INTERFACE I_MessageData

PROPERTY DirRoot : POINTER to string(255)
SET
END_SET
END_PROPERTY

PROPERTY ErrorIndex : reference to uint
SET
END_SET
END_PROPERTY

PROPERTY FileRoot : pointer to string(255)
SET
END_SET
END_PROPERTY

PROPERTY LocalTime : pointer to DT
SET
END_SET
END_PROPERTY

PROPERTY MessageIndex : reference to uint
SET
END_SET
END_PROPERTY

PROPERTY MsgList : pointer to ARRAY[1..GVL_MSG.MAX_MESSAGE] OF st_message
SET
END_SET
END_PROPERTY

END_INTERFACE

(* stored: Version 1.1.0.1
   Itf I_MessageData: Id {f6a96240-99ae-4618-b2ce-2104a304fee0}
   Property DirRoot: Id {caa07dbc-04ed-4392-a650-b335ab3d5005}
   Set Set: Id {fd0f934c-7d3d-4e0f-aecc-db828ecd61bd}
   Property ErrorIndex: Id {87d8f92c-f432-4c2d-b856-904c14d00dd3}
   Set Set: Id {18121a8a-40ab-41a6-b72d-61490f470a4a}
   Property FileRoot: Id {53c974bd-d010-4f69-a899-a1aaf707c45d}
   Set Set: Id {6ac54f9d-8006-4b91-9b1f-f40bcb34bbd2}
   Property LocalTime: Id {0ed9cddb-a9d3-4c4f-937d-34752c417a65}
   Set Set: Id {6a30d4b9-5ac5-49e6-828d-19fdd852b953}
   Property MessageIndex: Id {6bf976f6-99ce-4dda-b969-414b02b37e4d}
   Set Set: Id {06f307b0-f4e8-4091-b2ac-2535deb14a55}
   Property MsgList: Id {94d597a9-7a4f-47c6-8dfa-65040c34b4b7}
   Set Set: Id {2ea0ab99-0302-4fbc-b3e6-7665575ce24b} *)
